# EPICS substitutions: gigeApp/Db/pluginJPEG.substitutions
#
# pluginJPEG.substitutions
#

file NDPluginBase.template
{
	{
	P=$(CAM):,
	R=JPEG$(N):,
	PORT=JPEG$(N),
	ADDR=0,
	TIMEOUT=1,
	NDARRAY_PORT=$(PLUGIN_SRC),
	NDARRAY_ADDR=0
	}
}

file NDFile.template
{
	{
	P=$(CAM):,
	R=JPEG$(N):,
	PORT=JPEG$(N),
	ADDR=0,
	TIMEOUT=1
	}
}

file NDFileJPEG.template
{
	{
	P=$(CAM):,
	R=JPEG$(N):,
	PORT=JPEG$(N),
	ADDR=0,
	TIMEOUT=1
	}
}
